FUNCTION_BLOCK FB_RV_Ablaufsteuerung
VAR_IN_OUT
	Zustand			: ST_RV_Zustand;
	Stellwert			: ST_RV_Stellwert;
END_VAR
VAR_INPUT
	Steuerung		: ST_RV_Steuerung;
	Parameter		: ST_RV_Parameter;
END_VAR
VAR_OUTPUT
END_VAR
VAR
	Timer			: TON;
END_VAR

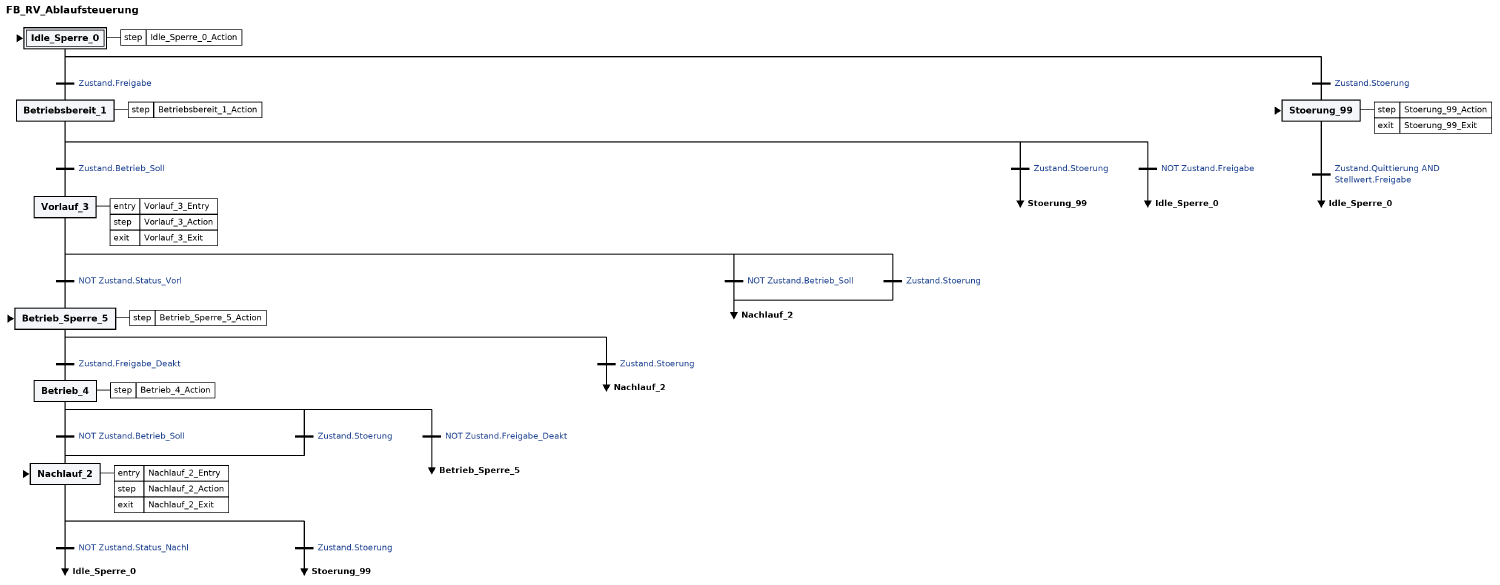
INITIAL_STEP Idle_Sperre_0:
    Idle_Sperre_0_Action(N);  // step action
END_STEP
TRANSITION FROM Idle_Sperre_0 TO Betriebsbereit_1
    := Zustand.Freigabe;
END_TRANSITION
TRANSITION FROM Idle_Sperre_0 TO Stoerung_99
    := Zustand.Stoerung;
END_TRANSITION
STEP Stoerung_99:
    Stoerung_99_Action(N);  // step action
    Stoerung_99_Exit(P0);  // exit action
END_STEP
TRANSITION FROM Stoerung_99 TO Idle_Sperre_0
    := Zustand.Quittierung AND Stellwert.Freigabe;
END_TRANSITION
STEP Betriebsbereit_1:
    Betriebsbereit_1_Action(N);  // step action
END_STEP
TRANSITION FROM Betriebsbereit_1 TO Vorlauf_3
    := Zustand.Betrieb_Soll;
END_TRANSITION
TRANSITION FROM Betriebsbereit_1 TO Stoerung_99
    := Zustand.Stoerung;
END_TRANSITION
TRANSITION FROM Betriebsbereit_1 TO Idle_Sperre_0
    := NOT Zustand.Freigabe;
END_TRANSITION
STEP Vorlauf_3:
    Vorlauf_3_Entry(P1);  // entry action
    Vorlauf_3_Action(N);  // step action
    Vorlauf_3_Exit(P0);  // exit action
END_STEP
TRANSITION FROM Vorlauf_3 TO Betrieb_Sperre_5
    := NOT Zustand.Status_Vorl;
END_TRANSITION
TRANSITION FROM Vorlauf_3 TO Nachlauf_2
    := NOT Zustand.Betrieb_Soll;
END_TRANSITION
TRANSITION FROM Vorlauf_3 TO Nachlauf_2
    := Zustand.Stoerung;
END_TRANSITION
STEP Betrieb_Sperre_5:
    Betrieb_Sperre_5_Action(N);  // step action
END_STEP
TRANSITION FROM Betrieb_Sperre_5 TO Betrieb_4
    := Zustand.Freigabe_Deakt;
END_TRANSITION
TRANSITION FROM Betrieb_Sperre_5 TO Nachlauf_2
    := Zustand.Stoerung;
END_TRANSITION
STEP Betrieb_4:
    Betrieb_4_Action(N);  // step action
END_STEP
TRANSITION FROM Betrieb_4 TO Nachlauf_2
    := NOT Zustand.Betrieb_Soll;
END_TRANSITION
TRANSITION FROM Betrieb_4 TO Nachlauf_2
    := Zustand.Stoerung;
END_TRANSITION
TRANSITION FROM Betrieb_4 TO Betrieb_Sperre_5
    := NOT Zustand.Freigabe_Deakt;
END_TRANSITION
STEP Nachlauf_2:
    Nachlauf_2_Entry(P1);  // entry action
    Nachlauf_2_Action(N);  // step action
    Nachlauf_2_Exit(P0);  // exit action
END_STEP
TRANSITION FROM Nachlauf_2 TO Idle_Sperre_0
    := NOT Zustand.Status_Nachl;
END_TRANSITION
TRANSITION FROM Nachlauf_2 TO Stoerung_99
    := Zustand.Stoerung;
END_TRANSITION

ACTION Betrieb_4_Action:
(* Stellwert setzen *)
Stellwert.Betrieb := TRUE;

(* Zustand setzen *)
Zustand.Betrieb	:= TRUE;
Zustand.Status := E_RV_Zustand_Status_Betrieb;
END_ACTION

ACTION Betrieb_Sperre_5_Action:
(* Stellwert setzen *)
Stellwert.Betrieb := TRUE;

(* Zustand setzen *)
Zustand.Betrieb	:= TRUE;
Zustand.Status := E_RV_Zustand_Status_Betrieb_Sperre;
END_ACTION

ACTION Betriebsbereit_1_Action:
(* Stellwert setzen *)
Stellwert.Betrieb := FALSE;


(* Zustand setzen *)
Zustand.Betrieb	:= FALSE;
Zustand.Status := E_RV_Zustand_Status_Betriebsbereit;
END_ACTION

ACTION Idle_Sperre_0_Action:
(* Stellwert setzen *)
Stellwert.Betrieb := FALSE;

(* Zustand setzen *)
Zustand.Betrieb	:= FALSE;
Zustand.Status := E_RV_Zustand_Status_Idle_Sperre;
END_ACTION

ACTION Nachlauf_2_Action:
(* Nachlauf Timer starten *)
Timer( 	IN := Zustand.Status_Nachl,
		PT := DINT_TO_TIME(Parameter.Zeit_Nachl)
);
Zustand.Status_Nachl	:= NOT(Timer.Q);

(* Stellwert setzen *)
Stellwert.Betrieb := FALSE;


(* Zustand setzen *)
Zustand.Betrieb	:= FALSE;
Zustand.Status := E_RV_Zustand_Status_Nachl;
END_ACTION

ACTION Nachlauf_2_Entry:
Zustand.Status_Nachl := TRUE;
(* Reset Timer *)
Timer(IN := FALSE);
END_ACTION

ACTION Nachlauf_2_Exit:
Zustand.Status_Nachl := FALSE;
END_ACTION

ACTION Stoerung_99_Action:
(* Stellwert setzen *)
Stellwert.Betrieb := FALSE;

(* Zustand setzen *)
Zustand.Stoerung := TRUE;
Zustand.Betrieb	:= FALSE;
Zustand.Status := E_RV_Zustand_Status_Stoerung;
END_ACTION

ACTION Stoerung_99_Exit:
Zustand.Stoerung	:= FALSE;
END_ACTION

ACTION Vorlauf_3_Action:
(* Vorlaufzeit Timer starten *)
Timer( 	IN := Zustand.Status_Vorl,
		PT := DINT_TO_TIME(Parameter.Zeit_Vorl)
);
Zustand.Status_Vorl := NOT (Timer.Q);

(* Stellwert setzen *)
Stellwert.Betrieb := TRUE;

(* Zustand setzen *)
Zustand.Betrieb	:= FALSE;
Zustand.Status := E_RV_Zustand_Status_Vorl;
END_ACTION

ACTION Vorlauf_3_Entry:
Zustand.Status_Vorl := TRUE;
(* Reset Timer *)
Timer(IN := FALSE);
END_ACTION

ACTION Vorlauf_3_Exit:
Zustand.Status_Vorl := FALSE;
END_ACTION

END_FUNCTION_BLOCK

(* stored: Version 1.1.0.1, ProductVersion 3.1.4024.9
   POU FB_RV_Ablaufsteuerung: Id {d3c69833-5af8-4002-9992-97e4c997f669}, SpecialFunc None
   Action Betrieb_4_Action: Id {4dfc20ad-ee75-4e1d-a334-e2b46a30a08d}
   Action Betrieb_Sperre_5_Action: Id {6123d587-ed44-4d3d-a402-6b00d571cbc4}
   Action Betriebsbereit_1_Action: Id {cab4f048-ba43-4a43-a8c8-1e76aee04278}
   Action Idle_Sperre_0_Action: Id {d997f80d-a2fe-46ef-9916-690853485029}
   Action Nachlauf_2_Action: Id {d5550e10-ab8e-4317-8d27-db23fd6c8456}
   Action Nachlauf_2_Entry: Id {cf82cf22-a872-49a1-a9bc-16054c475663}
   Action Nachlauf_2_Exit: Id {243e9ab8-b557-4861-9e3e-18266a9c9e55}
   Action Stoerung_99_Action: Id {5db58546-8fae-49a5-8c91-e18331209f1f}
   Action Stoerung_99_Exit: Id {4b7708c8-ae04-454e-ad9b-743145edb774}
   Action Vorlauf_3_Action: Id {52784732-5004-44dd-ab77-c59cc6504450}
   Action Vorlauf_3_Entry: Id {66877e60-4684-49d5-b55b-750afc964c50}
   Action Vorlauf_3_Exit: Id {97c03a86-37e4-485b-90ca-59cc24c7a91a} *)
